// SIMATIC S7-200 project (STEP 7-Micro/WIN), CPU 221 REL 01.10

SYMBOL_TABLE IO
电动缸负极限           I0.0     // 电动缸负极限
电动缸正极限           I0.1     // 电动缸正极限
电动缸原点            I0.2     // 电动缸原点
气压报警             I0.5     // 气压报警
光幕               I0.6     // 光幕
电动缸SRDY          I2.0     // 电动缸SRDY
电动缸STOP          I2.1     // 电动缸STOP
电动缸ALRM          I2.2     // 电动缸ALRM
涂胶监控             I2.4     // 涂胶监控
对射开关检测           I2.5     // 对射开关检测
防尘封在位检测          I2.6     // 急停按钮
急停按钮             I3.0     // 自动/手动
自动/手动            I3.1     // 复位按钮
复位按钮             I3.2     // 启动按钮
点胶启动按钮           I3.3     // 启动涂胶按钮
启动按钮             I3.4     // 点胶启动按钮
启动涂胶按钮           I3.5     // 电动缸脉冲指令
电动缸脉冲指令          Q0.0     // 电动缸方向指令
电动缸方向指令          Q0.1     // 电动缸上电
电动缸上电            Q0.6     // 电动缸SON
电动缸SON           Q2.0     // 电动缸CCLR
电动缸CCLR          Q2.1     // 电动缸ARST
电动缸ARST          Q2.2     // 电动缸EMGS
电动缸EMGS          Q2.3     // 涂脂1
涂脂1              Q3.0     // 涂脂2
压装涂脂2            Q3.1     // 点胶机上电
点胶机上电            Q3.2     // 点胶电机开
点胶电机开            Q3.3     // 红灯
红灯               Q3.4     // 黄灯
黄灯               Q3.5     // 绿灯
绿灯               Q3.6     // 蜂鸣器
蜂鸣器              Q3.7
END_SYMBOL_TABLE

SYMBOL_TABLE M3100
电动缸启动信号          M3110.0
电动缸工步号           MW3100
电动缸位置            MD3116
电动缸位置1           MD3120
电动缸位置2           MD3124
电动缸位置3           MD3128
电动缸位置4           MD3132
电动缸速度1           MD3152
电动缸速度2           MD3156
电动缸速度3           MD3160
电动缸速度4           MD3164
Tag_1            M3100.0
电动缸_运行中          M3110.1
电动缸_回原点信号        M3110.2
电动缸_回原点完成        M3110.3
电动缸_Reset启动      M3111.0
电动缸_Reset完成      M3111.1
电动缸_轴停止_启动       M3111.2
电动缸_轴停止_完成       M3111.3
电动缸_正转信号         M3111.4
电动缸_反转信号         M3111.5
电动缸_绝对值移动启动      M3112.0
电动缸_绝对值移动完成      M3112.1
电动缸_参数读取启动       M3112.2
电动缸_参数读取运行中      M3112.3
电动缸位置5           MD3136
电动缸位置6           MD3140
电动缸位置7           MD3144
电动缸速度            MD3148
电动缸速度5           MD3168
电动缸速度6           MD3172
电动缸速度7           MD3176
电动缸当前位置          MD3180
电动缸当前速度          MD3184
电动缸目标位置          MD3188
电动缸寸动速度          MD3196
电动缸启动信号1         M3113.0
电动缸启动信号2         M3113.1
电动缸启动信号3         M3113.2
电动缸启动信号4         M3113.3
电动缸启动信号5         M3113.4
电动缸完成信号1         M3114.0
电动缸完成信号2         M3114.1
电动缸完成信号3         M3114.2
电动缸完成信号4         M3114.3
电动缸完成信号5         M3114.4
M不合格提示按钮         M3106.0
涂脂自动工步号          MW3200
M涂脂1设定次数         MW3250
点胶自动工步号          MW3210
M压装位涂脂设定次数       MW3252
M涂脂1实际次数         MW3204
END_SYMBOL_TABLE

SYMBOL_TABLE M3000
流水线工步号           MW3000
产品类型             MW3002
RFID工步号          MW3004
芯片编号             MW3006
一键初始化工步号         MW3008
通讯状态             M3010.0
本工位合格            M3010.1
本工位完成            M3010.2
M涂脂1             M3020.0
上工位合格            M3030.0
上工位完成            M3030.1
联线状态             M3040.0
报警工步号            MW3050
员工权限             M3060.0
M压装位涂脂2          M3020.1
M点胶机开            M3020.2
M点胶机关            M3020.3
M点胶单循环           M3021.0
M涂脂单循环           M3021.1
M压装单循环           M3021.2
M单循环复位           M3021.3
本工位不合格           M3010.3
M光幕无效按钮          M3021.4
END_SYMBOL_TABLE
